FUNCTION_BLOCK AdsSocket
VAR_INPUT
	bEnable : BOOL;
END_VAR
VAR_OUTPUT
	PrgName : STRING; //descriptive string for the name of the running program, may or may not be used
	AmsNetId : T_AmsNetId;
	AmsPort : T_AmsPort; //for now, use ADS port 851 for communication
END_VAR
VAR_OUTPUT	
	receivingData : AdsData;
	sendingData : AdsData;
	
	readBusy : BOOL;
	readError : BOOL;
	readErrorId : UDINT;
	
	writeBusy : BOOL;
	writeError : BOOL;
	writeErrorId : UDINT;
	
	timeout : BOOL;
	busy : BOOL;
	error : BOOL;
	lastConnectedTime : TIMESTRUCT;
END_VAR
VAR	
	targetSocket : STRING := CONCAT('Sockets.', localPrgName); //write into the recipient's allocated socket for this system
	adsWriteSymbol : FB_WriteAdsSymByName;
	adsReadSymbol : FB_ReadAdsSymByName;
END_VAR
VAR	
	remoteFlag : BOOL; //receive FROM remote system
	localFlag : BOOL; //send TO remote system
	
	timer : TON;
	timerTrig : R_TRIG;
	
	flagWriter : FB_WriteAdsSymByName;
	nameWriter, netIdWriter, portWriter : FB_WriteAdsSymByName := (bWrite := FALSE);
	writeSync : BOOL := FALSE;
END_VAR
VAR_STAT
	localPrgName : STRING := TO_STRING(AreaNum.AREA_4);
	localAmsNetId : T_AmsNetId := '192.168.101.188.1.1';
	localAmsPort : T_AmsPort := 851;
END_VAR
(*
TCP-style ADS connection that only writes to a buffer in the recipient's AdsTcpUnit module
*)

targetSocket := CONCAT('Sockets.', localPrgName);
(*
IF NOT bEnable THEN
	RETURN;
END_IF
*)
setup();

flagSequence();

IF timeout THEN
	//stop data read/write attempts
	adsWriteSymbol.bWrite := FALSE;
	adsReadSymbol.bRead := FALSE;
ELSE
	//only writes if data has contents, otherwise remains false
	adsWriteSymbol.bWrite := NOT BufferIsEmpty(sendingData.binaryData) AND NOT adsWriteSymbol.bWrite;
END_IF

blocks();

METHOD PRIVATE blocks : BOOL
VAR_INPUT
END_VAR
adsReadSymbol(
	bRead:= , 
	sNetId:= AmsNetId, 
	nPort:= AmsPort, 
	sVarName:= , 
	nDestAddr:= , 
	nLen:= , 
	tTimeout:= , 
	eComMode:= , 
	bClearOnError:= , 
	bBusy=> readBusy, 
	bError=> readError, 
	nErrorId=> readErrorId);
	
adsWriteSymbol(
	bWrite:= , 
	sNetId:= AmsNetId, 
	nPort:= AmsPort, 
	sVarName:= CONCAT(targetSocket, '.receivingData'), 
	nSrcAddr:= ADR(sendingData), 
	nLen:= SIZEOF(sendingData), 
	tTimeout:= , 
	eComMode:= eAdsComModeSecureCom, 
	bBusy=> writeBusy, 
	bError=> writeError, 
	nErrorId=> writeErrorId);
	
IF NOT adsWriteSymbol.bBusy THEN
	MEMSET(ADR(sendingData), 0, SIZEOF(sendingData));
END_IF
END_METHOD

METHOD PRIVATE flagSequence : BOOL
VAR_INPUT
END_VAR
writeSync := NOT writeSync;

flagWriter(
	bWrite:= writeSync, 
	sNetId:= AmsNetId, 
	nPort:= AmsPort, 
	sVarName:= CONCAT(targetSocket, '.remoteFlag'), 
	nSrcAddr:= ADR(localFlag), 
	nLen:= SIZEOF(localFlag), 
	tTimeout:= , 
	eComMode:= , 
	bBusy=> busy, 
	bError=> error, 
	nErrorId=> );
	
timerTrig(
	CLK:= timerTrig.CLK XOR remoteFlag,
	Q=> ); //reset timer
	
IF timerTrig.Q THEN
	lastConnectedTime := MAIN.currentTime;
END_IF

timer(IN:= NOT timerTrig.Q, PT:= DEFAULT_ADS_TIMEOUT, Q=> timeout, ET=> );

IF NOT flagWriter.bBusy THEN
	localFlag := NOT localFlag;
END_IF
END_METHOD

METHOD send : BOOL
VAR_INPUT
	data : REFERENCE TO AdsData;
END_VAR
sendingData := data;
END_METHOD

METHOD PRIVATE setup : BOOL
VAR_INST
	name : STRING;
END_VAR
nameWriter(
	bWrite:= writeSync, 
	sNetId:= AmsNetId, 
	nPort:= AmsPort, 
	sVarName:= CONCAT(targetSocket, '.PrgName'), 
	nSrcAddr:= ADR(localPrgName), 
	nLen:= SIZEOF(localPrgName), 
	tTimeout:= , 
	eComMode:= , 
	bBusy=> busy, 
	bError=> error, 
	nErrorId=> );
	
netIdWriter(
	bWrite:= writeSync, 
	sNetId:= AmsNetId, 
	nPort:= AmsPort, 
	sVarName:= CONCAT(targetSocket, '.AmsNetId'), 
	nSrcAddr:= ADR(localAmsNetId), 
	nLen:= SIZEOF(localAmsNetId), 
	tTimeout:= , 
	eComMode:= , 
	bBusy=> , 
	bError=> , 
	nErrorId=> );
	
portWriter(
	bWrite:= writeSync, 
	sNetId:= AmsNetId, 
	nPort:= AmsPort, 
	sVarName:= CONCAT(targetSocket, '.AmsPort'), 
	nSrcAddr:= ADR(localAmsPort), 
	nLen:= SIZEOF(localAmsPort), 
	tTimeout:= , 
	eComMode:= , 
	bBusy=> , 
	bError=> , 
	nErrorId=> );
END_METHOD

END_FUNCTION_BLOCK

(* stored: Version 1.1.0.1, ProductVersion 3.1.4024.11
   POU AdsSocket: Id {4b08c35a-5e88-4e7b-a45b-894d0e3f10ba}, SpecialFunc None
   Method blocks: Id {aafa1f89-5424-428c-92a9-eff1fd826f0b}
   Method flagSequence: Id {282d8f86-2a36-4b14-910d-5c0d51c4379e}
   Method send: Id {17359b84-8e84-4f55-9ea9-7b9b4062b4aa}
   Method setup: Id {924e3658-3899-4767-999f-eb1a77052422} *)
